// TwinCAT 3 PLC project Refrigeration_Controller_Program
// ProgramVersion: 3.1.4024.0
// libraries:
//   Tc2_Standard, * (Beckhoff Automation GmbH)
//   Tc2_System, * (Beckhoff Automation GmbH)
//   Tc3_Module, * (Beckhoff Automation GmbH)
// project tree:
//   GVLs/ GVL_VAR.TcGVL
//   / PlcTask.TcTTO
//   POUs/ FB_Blinker.TcPOU, MAIN.TcPOU, Signals.TcPOU, Simulation.TcPOU

CONFIGURATION Refrigeration_Controller_Program
    RESOURCE PLC ON TwinCAT3
        TASK PlcTask(INTERVAL := T#10ms, PRIORITY := 20);
        PROGRAM MAIN WITH PlcTask : MAIN;
        PROGRAM Simulation WITH PlcTask : Simulation;
    END_RESOURCE
END_CONFIGURATION

// ---- GVLs/GVL_VAR.TcGVL
{attribute 'qualified_only'}
VAR_GLOBAL
	
	

	// Actual Temperature
	fTempActual: REAL := 0.5;
	// Set Temperature
	fTempSet: REAL := 0.2;
	// Door Status
	bDoorOpen: BOOL := FALSE;
	// Compressor Running Time After Which an Alarm Sounds
	tlmAlarmThreshold: TIME := T#30s;
	// Time from door opening after which alarm sounds
	tDoorOPenThreshold: TIME := T#10s;
	// Control Signal
	xCompressor: BOOL := FALSE;
	// Control Signal
	xSignal: BOOL := FALSE;
	// Status Message
	xLamp: BOOL := FALSE;
	// Ouput for controlling the compressor
	bCompressor: BOOL := FALSE;
	// Output for controlling signal
	bSingal: BOOL := FALSE;
	// Output for controlling the lamp
	bLamp: BOOL := FALSE;
END_VAR

// ---- POUs/MAIN.TcPOU
PROGRAM MAIN
VAR
	fHysteresis: REAL := 1;
	fbSR: SR;
END_VAR
VAR // added by the converter: edge detectors and wires of the graphical bodies
    _w1, _w2 : ANY;
END_VAR

fbSR(SET1 := _w1, RESET := _w2); // SR
GVL_VAR.bCompressor := fbSR.Q1;
_w1 := GVL_VAR.fTempActual > GVL_VAR.fTempSet + fHysteresis;
_w2 := GVL_VAR.fTempActual < GVL_VAR.fTempSet - fHysteresis;
Signals();

END_PROGRAM

// ---- POUs/Signals.TcPOU
PROGRAM Signals
VAR
	fbTimer1: TON;
	TON_0: TON;
END_VAR

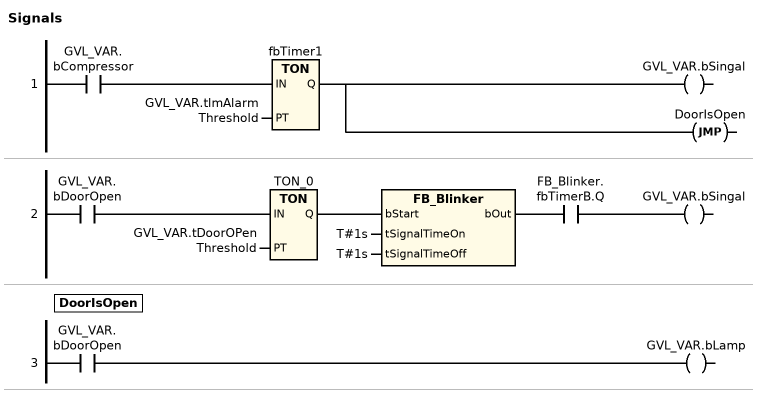
// NETWORK 1
fbTimer1(IN := GVL_VAR.bCompressor, PT := GVL_VAR.tlmAlarmThreshold); // TON
GVL_VAR.bSingal := fbTimer1.Q;
IF fbTimer1.Q THEN JMP DoorIsOpen; END_IF

// NETWORK 2
TON_0(IN := GVL_VAR.bDoorOpen, PT := GVL_VAR.tDoorOPenThreshold); // TON
FB_Blinker(bStart := TON_0.Q, tSignalTimeOn := T#1s, tSignalTimeOff := T#1s);
GVL_VAR.bSingal := FB_Blinker.bOut AND FB_Blinker.fbTimerB.Q;

// NETWORK 3
DoorIsOpen:
GVL_VAR.bLamp := GVL_VAR.bDoorOpen;

END_PROGRAM

// ---- POUs/FB_Blinker.TcPOU
PROGRAM FB_Blinker
VAR
	fbTimerA: TON;
	fbTimerB: TON;
END_VAR

VAR_INPUT
	bStart: BOOL;
	tSignalTimeOn: TIME;
	tSignalTimeOff: TIME;
END_VAR
VAR_OUTPUT
	bOut: BOOL;
END_VAR

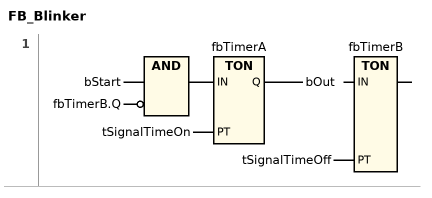
// NETWORK 1
fbTimerA(IN := bStart AND NOT fbTimerB.Q, PT := tSignalTimeOn); // TON
bOut := fbTimerA.Q;
fbTimerB(IN := fbTimerA.Q, PT := tSignalTimeOff); // TON

END_PROGRAM

// ---- POUs/Simulation.TcPOU
PROGRAM Simulation
VAR
	fbT1 : TON; //The temperature is decreased on a time delay, when the compressor has been activated
	tCooling : TIME := T#500MS; 
	bReduceTemp : BOOL;//Signal for decreasing the temperature
	fbT2 : TON; //The temperature is increased on a time delay, when the compressor has been deactivated
	tEnvironment : TIME := T#2S; //Delay time when the door is closed
	tEnvironmentDoorOpen : TIME := T#1S; //Delay time when the door is opened
	bRaiseTemp : BOOL; //Signal for increasing the temperature
	tImTemp : TIME; //Delay time
	nCounter : INT;
END_VAR

//After the compressor has been activated due to fTempActual being above the setpoint plus hysteresis, the temperature decreases
//The temperature is decremented by 0.1 degree Celsius per cycle after a delay of P_Cooling

IF GVL_VAR.bCompressor THEN
	fbT1(IN:=GVL_VAR.bCompressor, PT := tCooling, Q => bReduceTemp);
	IF bReduceTemp THEN
		GVL_VAR.fTempActual := GVL_VAR.fTempActual - 0.1;
		fbT1(IN:= FALSE);
	END_IF
END_IF

//If the door is open, the warning will occur faster; SEL selects tEnvironmentDoorOpen

tImTemp := SEL(GVL_VAR.bDoorOpen, tEnvironment, tEnvironmentDoorOpen);

//If the compressor is not in operation the cooling chamber must start heating up again
//The temperature is incremented by 0.1 degrees per cycle after a delay of tImTemp

fbT2(IN:= TRUE, PT:= tImTemp, Q=> bRaiseTemp);
IF bRaiseTemp THEN
	GVL_VAR.fTempActual := GVL_VAR.fTempActual + 0.1;
	fbT2(IN:=FALSE); //this resets the timer by taking the input LOW
END_IF

END_PROGRAM
